// TIA Portal V20 export
DATA_BLOCK "GLOBAL_Axis_HMI_IF_DB"   // DB202
{ S7_Optimized_Access := 'TRUE' }
// stored: AutoNumber false, MemoryReserve 100
   VAR RETAIN
      Axis { S7_SetPoint := 'True'} : Array[0..10] of "Axis_IF_HMI";
   END_VAR
BEGIN
END_DATA_BLOCK
